FUNCTION_BLOCK csvParser (* filenames output *)
  (* Version 1.0, AN, SWDC RTSoft *)
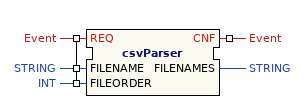
  EVENT_INPUT
    REQ WITH FILENAME, FILEORDER;
  END_EVENT
  EVENT_OUTPUT
    CNF WITH STATUS;
  END_EVENT
  VAR_INPUT
    FILENAME : STRING;
    FILEORDER : INT;
  END_VAR
  VAR_OUTPUT
    FILENAMES : STRING;
  END_VAR
END_FUNCTION_BLOCK
